// TIA Portal V18 export
FUNCTION "InputMapping" : Void   // FC1, LAD
TITLE = Input Mapping
{ S7_Optimized_Access := 'TRUE' }
VERSION : 0.1
// Input and HMI
// stored: AutoNumber true, IsIECCheckEnabled false, SetENOAutomatically false, UDAEnableTagReadback false
BEGIN

REGION Network 1: Input Control Button AGV - Betriebsarten
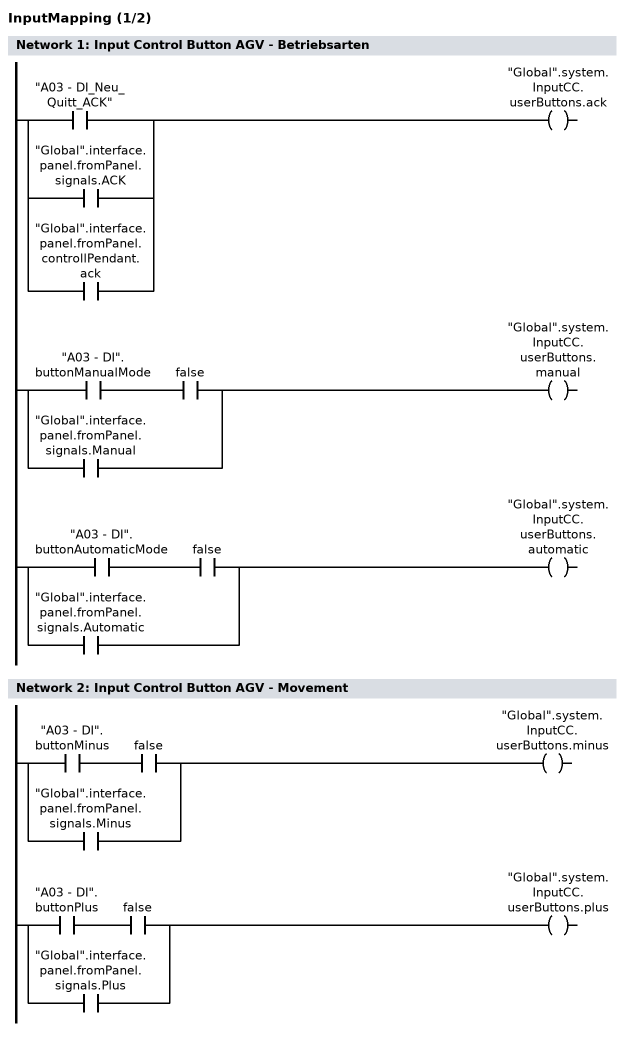
   RUNG wire#powerrail
      Contact( "A03 - DI_Neu_Quitt_ACK" )
      wire#w1
      Coil( "Global".system.InputCC.userButtons.ack )
   END_RUNG
   RUNG wire#powerrail
      Contact( "Global".interface.panel.fromPanel.signals.ACK )
   END_RUNG wire#w1
   RUNG wire#powerrail
      Contact( "Global".interface.panel.fromPanel.controllPendant.ack )
   END_RUNG wire#w1
   RUNG wire#powerrail
      Contact( "A03 - DI".buttonManualMode )
      Contact( false )
      wire#w2
      Coil( "Global".system.InputCC.userButtons.manual )
   END_RUNG
   RUNG wire#powerrail
      Contact( "Global".interface.panel.fromPanel.signals.Manual )
   END_RUNG wire#w2
   RUNG wire#powerrail
      Contact( "A03 - DI".buttonAutomaticMode )
      Contact( false )
      wire#w3
      Coil( "Global".system.InputCC.userButtons.automatic )
   END_RUNG
   RUNG wire#powerrail
      Contact( "Global".interface.panel.fromPanel.signals.Automatic )
   END_RUNG wire#w3
   // the same network as SCL:
   "Global".system.InputCC.userButtons.ack := "A03 - DI_Neu_Quitt_ACK" OR "Global".interface.panel.fromPanel.signals.ACK OR "Global".interface.panel.fromPanel.controllPendant.ack;
   "Global".system.InputCC.userButtons.manual := ("A03 - DI".buttonManualMode AND false) OR "Global".interface.panel.fromPanel.signals.Manual;
   "Global".system.InputCC.userButtons.automatic := ("A03 - DI".buttonAutomaticMode AND false) OR "Global".interface.panel.fromPanel.signals.Automatic;
END_REGION

REGION Network 2: Input Control Button AGV - Movement
   RUNG wire#powerrail
      Contact( "A03 - DI".buttonMinus )
      Contact( false )
      wire#w1
      Coil( "Global".system.InputCC.userButtons.minus )
   END_RUNG
   RUNG wire#powerrail
      Contact( "Global".interface.panel.fromPanel.signals.Minus )
   END_RUNG wire#w1
   RUNG wire#powerrail
      Contact( "A03 - DI".buttonPlus )
      Contact( false )
      wire#w2
      Coil( "Global".system.InputCC.userButtons.plus )
   END_RUNG
   RUNG wire#powerrail
      Contact( "Global".interface.panel.fromPanel.signals.Plus )
   END_RUNG wire#w2
   // the same network as SCL:
   "Global".system.InputCC.userButtons.minus := ("A03 - DI".buttonMinus AND false) OR "Global".interface.panel.fromPanel.signals.Minus;
   "Global".system.InputCC.userButtons.plus := ("A03 - DI".buttonPlus AND false) OR "Global".interface.panel.fromPanel.signals.Plus;
END_REGION

REGION Network 3: Input Control Button AGV - Test
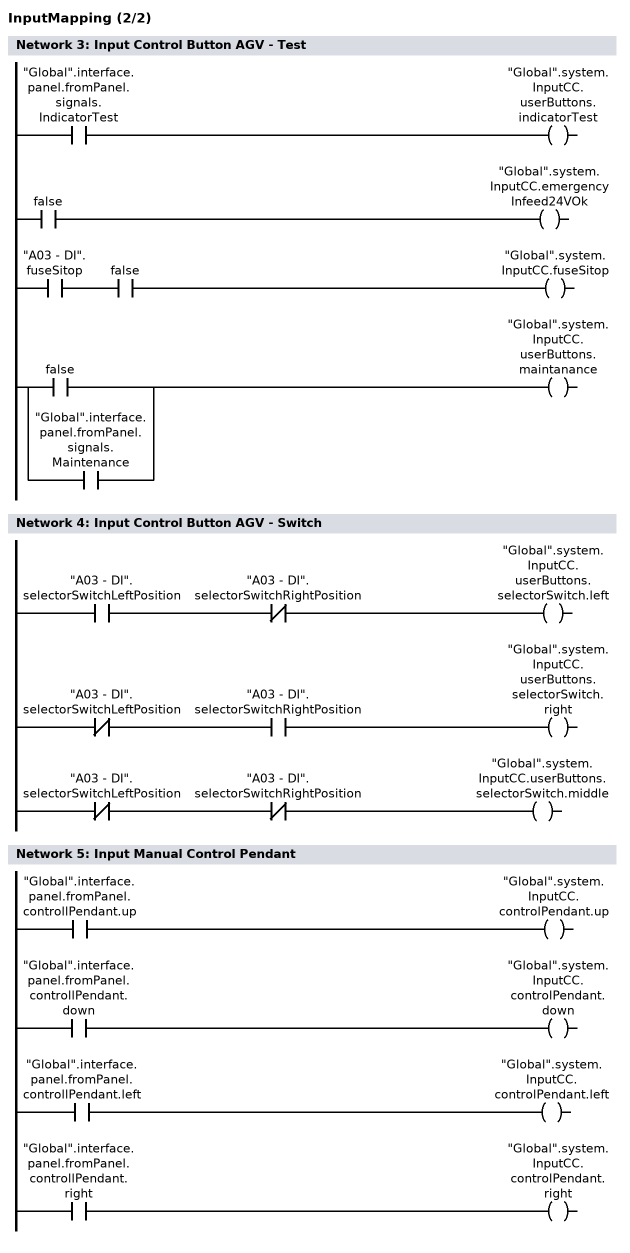
   RUNG wire#powerrail
      Contact( "Global".interface.panel.fromPanel.signals.IndicatorTest )
      Coil( "Global".system.InputCC.userButtons.indicatorTest )
   END_RUNG
   RUNG wire#powerrail
      Contact( false )
      Coil( "Global".system.InputCC.emergencyInfeed24VOk )
   END_RUNG
   RUNG wire#powerrail
      Contact( "A03 - DI".fuseSitop )
      Contact( false )
      Coil( "Global".system.InputCC.fuseSitop )
   END_RUNG
   RUNG wire#powerrail
      Contact( false )
      wire#w1
      Coil( "Global".system.InputCC.userButtons.maintanance )
   END_RUNG
   RUNG wire#powerrail
      Contact( "Global".interface.panel.fromPanel.signals.Maintenance )
   END_RUNG wire#w1
   // the same network as SCL:
   "Global".system.InputCC.userButtons.indicatorTest := "Global".interface.panel.fromPanel.signals.IndicatorTest;
   "Global".system.InputCC.emergencyInfeed24VOk := false;
   "Global".system.InputCC.fuseSitop := "A03 - DI".fuseSitop AND false;
   "Global".system.InputCC.userButtons.maintanance := false OR "Global".interface.panel.fromPanel.signals.Maintenance;
END_REGION

REGION Network 4: Input Control Button AGV - Switch
   RUNG wire#powerrail
      Contact( "A03 - DI".selectorSwitchLeftPosition )
      I_Contact( "A03 - DI".selectorSwitchRightPosition )
      Coil( "Global".system.InputCC.userButtons.selectorSwitch.left )
   END_RUNG
   RUNG wire#powerrail
      I_Contact( "A03 - DI".selectorSwitchLeftPosition )
      Contact( "A03 - DI".selectorSwitchRightPosition )
      Coil( "Global".system.InputCC.userButtons.selectorSwitch.right )
   END_RUNG
   RUNG wire#powerrail
      I_Contact( "A03 - DI".selectorSwitchLeftPosition )
      I_Contact( "A03 - DI".selectorSwitchRightPosition )
      Coil( "Global".system.InputCC.userButtons.selectorSwitch.middle )
   END_RUNG
   // the same network as SCL:
   "Global".system.InputCC.userButtons.selectorSwitch.left := "A03 - DI".selectorSwitchLeftPosition AND NOT "A03 - DI".selectorSwitchRightPosition;
   "Global".system.InputCC.userButtons.selectorSwitch.right := NOT "A03 - DI".selectorSwitchLeftPosition AND "A03 - DI".selectorSwitchRightPosition;
   "Global".system.InputCC.userButtons.selectorSwitch.middle := NOT "A03 - DI".selectorSwitchLeftPosition AND NOT "A03 - DI".selectorSwitchRightPosition;
END_REGION

REGION Network 5: Input Manual Control Pendant
   RUNG wire#powerrail
      Contact( "Global".interface.panel.fromPanel.controllPendant.up )
      Coil( "Global".system.InputCC.controlPendant.up )
   END_RUNG
   RUNG wire#powerrail
      Contact( "Global".interface.panel.fromPanel.controllPendant.down )
      Coil( "Global".system.InputCC.controlPendant.down )
   END_RUNG
   RUNG wire#powerrail
      Contact( "Global".interface.panel.fromPanel.controllPendant.left )
      Coil( "Global".system.InputCC.controlPendant.left )
   END_RUNG
   RUNG wire#powerrail
      Contact( "Global".interface.panel.fromPanel.controllPendant.right )
      Coil( "Global".system.InputCC.controlPendant.right )
   END_RUNG
   // the same network as SCL:
   "Global".system.InputCC.controlPendant.up := "Global".interface.panel.fromPanel.controllPendant.up;
   "Global".system.InputCC.controlPendant.down := "Global".interface.panel.fromPanel.controllPendant.down;
   "Global".system.InputCC.controlPendant.left := "Global".interface.panel.fromPanel.controllPendant.left;
   "Global".system.InputCC.controlPendant.right := "Global".interface.panel.fromPanel.controllPendant.right;
END_REGION
END_FUNCTION
